TYPE "PPrf_Data"
VERSION : 0.1
// Block: PPrf_Data
   STRUCT
      Header : Prg_Header;
      GeneralData : PPrf_Generic;
      SetUp : PPrf_SetUp;
      A01_CoilHandling : PPrf_CoilHandlig;
      A02_1_PartsCutting : PPrf_A02_S1_PartsCutting;
      A0301_A0302 : PPrf_A0301_0302_Assemblaggio;
      A0303_A0304 : PPrf_A0304_0304_Scarico;
   END_STRUCT;

END_TYPE
